(* PLC project CoDeSys External Library Template, WAGO e!COCKPIT e!COCKPIT, author 3S - Smart Software Solutions GmbH *)
(* stored: creationDateTime 2019-10-29T12:22:40.9371025, version 3.5.5.30, modificationDateTime 2019-10-24T14:40:07.960949, organization 3S - Smart Software Solutions GmbH *)
(* Library project template with all possible element types, docu and a sample project structure *)

FUNCTION fnKonwersja512na4x128 : BOOL
  VAR_INPUT
    sKomunikat512 : alSTRINGKomunikat;
  END_VAR
  VAR_IN_OUT
    sKomunikatCzesc1 : STRING(128);
    sKomunikatCzesc2 : STRING(128);
    sKomunikatCzesc3 : STRING(128);
    sKomunikatCzesc4 : STRING(128);
  END_VAR

            sKomunikatCzesc1 := MID(sKomunikat512 , 128 , 1);
sKomunikatCzesc2 := MID(sKomunikat512 , 128 , 129);
sKomunikatCzesc3 := MID(sKomunikat512 , 128 , 513);
sKomunikatCzesc4 := MID(sKomunikat512 , 128 , 385);
fnKonwersja512na4x128 := TRUE;

          
END_FUNCTION
